// TIA Portal V19 export
DATA_BLOCK "CarriageLub_PERS"   // DB131
// stored: MemoryReserve 100
   VAR RETAIN
      Carriage_SlideLubr : Struct
         Control : "LubrValve_Pers";
         EvLub { S7_SetPoint := 'True'} : "LubrPump_Par";
      END_STRUCT;
   END_VAR
   VAR
      CarriageLub_Pers_HMI_ResetCounter : Bool := FALSE;
   END_VAR
BEGIN
   Carriage_SlideLubr.Control.Par.SystemOn := TRUE;
   Carriage_SlideLubr.Control.Par.EnableCheckFdbk := FALSE;
   Carriage_SlideLubr.Control.Par.CycleFdbkCheckTime := T#0MS;
   Carriage_SlideLubr.Control.Par.WorkTime := T#0MS;
   Carriage_SlideLubr.Control.Par.ValveONTime := T#0MS;
   Carriage_SlideLubr.Control.Par.ValveOFFTime := T#8S;
   Carriage_SlideLubr.Control.Par.ValvePumpSetPoint := 3;
   Carriage_SlideLubr.Control.Par.LubrReqSetPoint := 400.0;
   Carriage_SlideLubr.Control.ValvePumpCounter := 2;
   Carriage_SlideLubr.Control.LubrReqCounter := 312.596580000482;
   Carriage_SlideLubr.EvLub.LowLevelCheckTime := T#10S;
   Carriage_SlideLubr.EvLub.ValveONTime := T#1S;
   Carriage_SlideLubr.EvLub.ValveOFFTime := T#3S;
END_DATA_BLOCK
